TYPE stEcSlaveState :
STRUCT
	ERROR		: BOOL;
	Init 		: BOOL;
	PROCESSING 	: BOOL;
	OP          : BOOL;
	
END_STRUCT
END_TYPE

(* stored: Version 1.1.0.1, ProductVersion 3.1.4024.12
   DUT stEcSlaveState: Id {c02ab940-f675-4b92-952a-150a754cb782} *)
